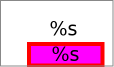
VISUALIZATION Obj_PDU_Breaker  // 114x67
VAR_INPUT
	sIndex : STRING;
	bClosed : BOOL;
	bOffline : BOOL;
	bHealthy : BOOL;
END_VAR
    Rectangle (27,42 77x25), "%s", colour toggle: bClosed, text list: 'PDU_Breaker_Status', text index: bClosed
    Rectangle (13,16 101x26), "%s", text variable: sIndex
    Rectangle (27,42 77x25), "%s", invisible if: not bOffline, text list: 'PDU_Breaker_Status', text index: bClosed
    Rectangle (27,42 77x25), invisible if: bHealthy
END_VISUALIZATION

(* stored: Version 1.1.0.1, ProductVersion 3.1.4024.12
   Visu Obj_PDU_Breaker: Id {1adff825-0957-41c3-a732-13479bda54c7} *)
